FUNCTION_BLOCK FB_NormalAlarmProfile IMPLEMENTS I_AlarmProfile
VAR
	
END_VAR

METHOD GetName  : STRING
VAR_INPUT
END_VAR
GetName := 'NORMAL';
END_METHOD

METHOD GetVoteAlert : INT
VAR_INPUT
END_VAR
GetVoteAlert     := GVL_SafetyLimits.c_nVOTE_ALERT;      // 1
END_METHOD

METHOD GetVoteEmergency : INT
VAR_INPUT
END_VAR
GetVoteEmergency := GVL_SafetyLimits.c_nVOTE_EMERGENCY;  // 3
END_METHOD

METHOD GetVoteWarning  : INT
VAR_INPUT
END_VAR

GetVoteWarning   := GVL_SafetyLimits.c_nVOTE_WARNING;    // 2
END_METHOD

END_FUNCTION_BLOCK

(* stored: Version 1.1.0.1, ProductVersion 3.1.4024.16
   POU FB_NormalAlarmProfile: Id {97e8a250-2a37-4dfd-98bd-fb2fcd10613b}, SpecialFunc None
   Method GetName: Id {2ba4b09d-f7a3-47ee-b781-65fd41351279}
   Method GetVoteAlert: Id {9f334bf8-4435-42ad-b608-b62d0b8e9456}
   Method GetVoteEmergency: Id {de5a0f29-02d6-4f17-ac4a-522c268954b2}
   Method GetVoteWarning: Id {e314dfc0-87eb-4281-a379-954c1f51ecec} *)
